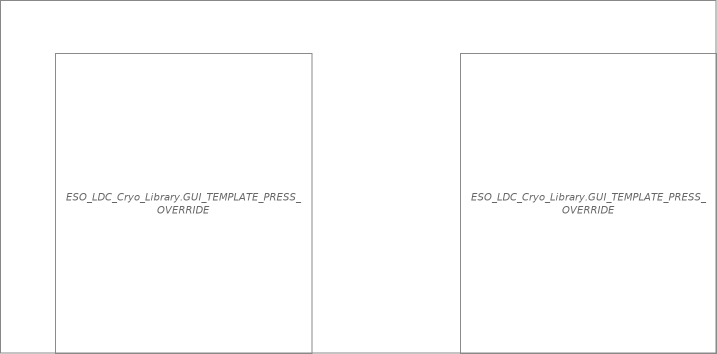
VISUALIZATION VISU_NOTT_PRESSURES  // 717x354
    Frame (55,53 257x301)
        shows ESO_LDC_Cryo_Library.GUI_TEMPLATE_PRESS_OVERRIDE(m_Cmd := MAIN.nott_cryo_ctrl.ctrl.por_VAGC, m_Press := MAIN.nott_cryo_ctrl.VAGC)
    Frame (460,53 257x301)
        shows ESO_LDC_Cryo_Library.GUI_TEMPLATE_PRESS_OVERRIDE(m_Cmd := MAIN.nott_cryo_ctrl.ctrl.por_HPG, m_Press := MAIN.nott_cryo_ctrl.HPG)
END_VISUALIZATION

(* stored: Version 1.1.0.1, ProductVersion 3.1.4026.18
   Visu VISU_NOTT_PRESSURES: Id {40ab7661-4c70-4963-a3cc-98ecc35ec19c} *)
